# B&R Automation Studio project A2019059_Linka_Power_CP (part 58)

#### Main.st - Init, cyclic, exit code
```iecst
PROGRAM _INIT
	(* Insert code here *)

END_PROGRAM

PROGRAM _CYCLIC

	//Volanie funkcie SequenceControl//
	SequenceControl(SC:= SC_Devlink);

    //Mapovanie premenných//
    FTP_DMP_CAM17.STATUS.CisloPoruchy:= CisloAlarmu;
    FTP_DMP_CAM17.STATUS.AdresarPrazdny:= AdresarPrazdny;

    //Čísla alarmov//
    //1 - porucha otvorenia komunikacie z adresarom PLC
    //2 - porucha otvorenia komunikacie z adresarom Panasonic
    //3 - porucha načítania adresára kamery
    //4 - porucha zápisu najdených súborov
    //5 - porucha premenovania fotky
    //6 - porucha vytvorenia adresara na disku Panasonic
    //7 - porucha kopirovania fotky na server Panasonic
    //8 - porucha vymazania fotky v adresari kamery

    CASE SC_Devlink.Step OF

        0:
            SC_Devlink.StepName:= '0 - Nulovanie';
            FTP_DMP_CAM17.STATUS.KomunikaciaError:= FALSE;
            FTP_DMP_CAM17.STATUS.KomunikaciaUkoncena:= FALSE;
            PocetHladaniFotky:= 0;
            AdresarPrazdny:= FALSE;
            PocetNajdenychSuborov:= 0;
            PocetNajdenychAdresarov:= 0;
            PocetPremenovanychSuborov:= 1;
            PocetSkopirovanychSuborov:= 1;
            PocetVymazanychSuborov:= 1;
            i:= 0;
            SC_Devlink.Step:= 1;

        1:
            SC_Devlink.StepName:= '1 - Rozhodnutie o cinnosti';
            IF FTP_DMP_CAM17.CMD.OdosliFotku THEN
                CisloAlarmu:= 0;
                SC_Devlink.Step:= 10;
            ELSIF FTP_DMP_CAM17.CMD.VymazFotku THEN
                CisloAlarmu:= 0;
                SC_Devlink.Step:= 150;
            END_IF

        10:
            SC_Devlink.StepName:= '10 - Skopirovanie fotky do adresara DMP, otvorenie komunikacie z adresarom PLC';
            SC_Devlink.IdleTime.PT:= T#3s;
            SC_Devlink.AlarmTime.PT:= T#3s;

            DevLink_0.enable:= TRUE;
            DevLink_0.pDevice:= ADR('CAM17');
            DevLink_0.pParam:= ADR('/SIP=192.168.122.3 /PROTOCOL=ftp /USER=cam17 /PASSWORD=.cam17');
            DevLink_0();

            IF DevLink_0.enable THEN
                IF DevLink_0.status = 0 THEN
                    ID_Adresara1:= DevLink_0.handle;
                    SC_Devlink.ResetStep:= TRUE;
                    SC_Devlink.Step:= 15;//15
                ELSIF DevLink_0.status = 20730 THEN
                    ID_Adresara1:= DevLink_0.handle;
                    SC_Devlink.ResetStep:= TRUE;
                    SC_Devlink.Step:= 15;//15
                ELSIF DevLink_0.status = 65535 THEN
                    //BUSY//
                ELSE
                    CisloAlarmu:= 1;
                    FTP_DMP_CAM17.STATUS.KomunikaciaError:= TRUE;
                    SC_Devlink.ResetStep:= TRUE;
                    SC_Devlink.Step:= 13;
                END_IF
            END_IF

        13: SC_Devlink.StepName:= '13 - Skopirovanie fotky do adresara DMP, odpojenie od adresara PLC';
            SC_Devlink.IdleTime.PT:= T#3s;
            SC_Devlink.AlarmTime.PT:= T#3s;

            DevUnlink_0.enable:= TRUE;
            DevUnlink_0.handle:= ID_Adresara1;
            DevUnlink_0();

            IF DevUnlink_0.enable THEN
                IF DevUnlink_0.status = 0 THEN
                    SC_Devlink.ResetStep:= TRUE;
                    SC_Devlink.Step:= 100;
                ELSIF DevUnlink_0.status = 20731 THEN
                    SC_Devlink.ResetStep:= TRUE;
                    SC_Devlink.Step:= 100;
                ELSIF DevUnlink_0.status = 65535 THEN
                    //BUSY//
                ELSE
                    SC_Devlink.ResetStep:= TRUE;
                    SC_Devlink.Step:= 100;
                END_IF
            END_IF

        15:
            SC_Devlink.StepName:= '15 - Skopirovanie fotky do adresara DMP, otvorenie komunikacie z adresarom DMP';
            SC_Devlink.IdleTime.PT:= T#3s;
            SC_Devlink.AlarmTime.PT:= T#3s;

            DevLink_1.enable:= TRUE;
            DevLink_1.pDevice:= ADR('DMP_CAM17');
            DevLink_1.pParam:= ADR('/SIP=192.168.122.3 /PROTOCOL=ftp /USER=dmp_cam17 /PASSWORD=.dmp_cam17');
            DevLink_1();

            IF DevLink_1.enable THEN
                IF DevLink_1.status = 0 THEN
                    ID_Adresara2:= DevLink_0.handle;
                    SC_Devlink.ResetStep:= TRUE;
                    SC_Devlink.Step:= 20;
                ELSIF DevLink_1.status = 20730 THEN
                    ID_Adresara2:= DevLink_1.handle;
                    SC_Devlink.ResetStep:= TRUE;
                    SC_Devlink.Step:= 20;
                ELSIF DevLink_1.status = 65535 THEN
                    //BUSY//
                ELSE
                    CisloAlarmu:= 2;
                    FTP_DMP_CAM17.STATUS.KomunikaciaError:= TRUE;
                    SC_Devlink.ResetStep:= TRUE;
                    SC_Devlink.Step:= 18;
                END_IF
            END_IF

        18: SC_Devlink.StepName:= '18 - Skopirovanie fotky do adresara DMP, odpojenie od adresara DMP';
            SC_Devlink.IdleTime.PT:= T#3s;
            SC_Devlink.AlarmTime.PT:= T#3s;

            DevUnlink_1.enable:= TRUE;
            DevUnlink_1.handle:= ID_Adresara2;
            DevUnlink_1();

            IF DevUnlink_1.enable THEN
                IF DevUnlink_1.status = 0 THEN
                    SC_Devlink.ResetStep:= TRUE;
                    SC_Devlink.Step:= 100;
                ELSIF DevUnlink_1.status = 20731 THEN
                    SC_Devlink.ResetStep:= TRUE;
                    SC_Devlink.Step:= 100;
                ELSIF DevUnlink_1.status = 65535 THEN
                    //BUSY//
                ELSE
                    SC_Devlink.ResetStep:= TRUE;
                    SC_Devlink.Step:= 100;
                END_IF
            END_IF

        20:	SC_Devlink.StepName:= '20 - Skopirovanie fotky do adresara DMP, nacitanie adresara pred kopirovanim fotiek na server Panasonic';
            SC_Devlink.IdleTime.PT:= T#3s;
            SC_Devlink.AlarmTime.PT:= T#3s;

            DirInfo_0.enable:= TRUE;
            DirInfo_0.pDevice:= ADR('CAM17');
            DirInfo_0.pPath:= ADR('/');   //ak je nula tak číta všetky súbory a adresáre v koreni ak je "/Temp" tak číta všetky súbory a adresáre v adresári Temp//
            DirInfo_0();

            IF DirInfo_0.status = 0 THEN
                PocetNajdenychAdresarov:= DirInfo_0.dirnum;
                PocetNajdenychSuborov:= DirInfo_0.filenum;
                brsmemset(ADR(FileList[0]),0, SIZEOF(FileList));  //Vynulovanie pola stringov pre záznam adresárov a súborov
                SC_Devlink.ResetStep:= TRUE;
                SC_Devlink.Step:= 45;
            ELSIF DirInfo_0.status = 65535 THEN
                //BUSY//
            ELSIF DirInfo_0.status = 20723 THEN
                CisloAlarmu:= 3;
                FTP_DMP_CAM17.STATUS.KomunikaciaError:= TRUE;
                SC_Devlink.ResetStep:= TRUE;
                SC_Devlink.Step:= 100;
            ELSE
                CisloAlarmu:= 3;
                FTP_DMP_CAM17.STATUS.KomunikaciaError:= TRUE;
                SC_Devlink.ResetStep:= TRUE;
                SC_Devlink.Step:= 100;
            END_IF

        45: SC_Devlink.StepName:= '45 - Skopirovanie fotky do adresara DMP, zapis nazvou najdenych suborov do pola stringov';
            SC_Devlink.IdleTime.PT:= T#3s;
            SC_Devlink.AlarmTime.PT:= T#3s;

            DirRead_0.enable:= TRUE;
            DirRead_0.pDevice:= ADR('CAM17');
            DirRead_0.pPath:= ADR('/');   //ak je nula tak číta všetky súbory a adresáre v koreni ak je "/Temp" tak číta všetky súbory a adresáre v adresári Temp//
            DirRead_0.option:= fiFILE; //Zapíše súbory aj adresáre, ak je fiDIRECTORY zapíše len adresáre, ak je fiFILE tak zapíše len súbory//
            DirRead_0.entry:= i; //index zapisovania do pola//
            DirRead_0.pData:= ADR(ReadData);
            DirRead_0.data_len:= SIZEOF(ReadData);
            DirRead_0();

            IF DirRead_0.status = 0 THEN
                brsstrcpy(ADR(FileList[i]), ADR(ReadData.Filename[0])); //Uloženie názvou adresárov a súborov do pola stringov
                IF i< 100 THEN
                    i:= i + 1;
                END_IF
            ELSIF DirRead_0.status = 20702 THEN
                i:= 0;
                SC_Devlink.ResetStep:= TRUE;
                SC_Devlink.Step:= 48;
            ELSIF DirRead_0.status = 65535 THEN
                //BUSY//
            ELSE
                CisloAlarmu:= 4;
                FTP_DMP_CAM17.STATUS.KomunikaciaError:= TRUE;
                SC_Devlink.ResetStep:= TRUE;
                SC_Devlink.Step:= 100;
            END_IF

        48: SC_Devlink.StepName:= '48 - Skopirovanie fotky do adresara DMP, kopirovanie fotky do adresara DMP';
            SC_Devlink.IdleTime.PT:= T#3s;
            SC_Devlink.AlarmTime.PT:= T#3s;

            ZdrojKopirovaniaSuboru:= '';
            brsstrcat(ADR(ZdrojKopirovaniaSuboru),ADR('/'));
            brsstrcat(ADR(ZdrojKopirovaniaSuboru),ADR(FileList[i]));

            CielKopirovaniaSuboru:= '';
            brsstrcat(ADR(CielKopirovaniaSuboru),ADR('/'));
            brsstrcat(ADR(CielKopirovaniaSuboru),ADR(FileList[i]));

            FileCopy_0.enable:= TRUE;
            FileCopy_0.pSrcDev:= ADR('CAM17'); //Zdrojové zariadenie od kial sa kopíruje
            FileCopy_0.pSrc:= ADR(ZdrojKopirovaniaSuboru);
            FileCopy_0.pDestDev:= ADR('DMP_CAM17'); //Cielové zariadenie kam sa má súbor skopírovať
            FileCopy_0.pDest:= ADR(CielKopirovaniaSuboru);
            FileCopy_0();

            IF FileCopy_0.status = 0 THEN
                SC_Devlink.ResetStep:= TRUE;
                SC_Devlink.Step:= 50;
            ELSIF FileCopy_0.status = 65535 THEN
                //BUSY//
            ELSIF FileCopy_0.status = 20705 THEN
                SC_Devlink.ResetStep:= TRUE;
                SC_Devlink.Step:= 50;
            ELSIF FileCopy_0.status = 20708 THEN
                AdresarPrazdny:= TRUE;
                FTP_DMP_CAM17.STATUS.KomunikaciaUkoncena:= TRUE;
                SC_Devlink.ResetStep:= TRUE;
                SC_Devlink.Step:= 100;
            ELSE
                CisloAlarmu:= 7;
                FTP_DMP_CAM17.STATUS.KomunikaciaError:= TRUE;
                SC_Devlink.ResetStep:= TRUE;
                SC_Devlink.Step:= 100;
            END_IF

        50: SC_Devlink.StepName:= '50 - Skopirovanie fotky do adresara DMP, kontrola poctu skopirovanych suborov';
            SC_Devlink.IdleTime.PT:= T#3s;
            SC_Devlink.AlarmTime.PT:= T#3s;

            IF PocetSkopirovanychSuborov < PocetNajdenychSuborov THEN
                PocetSkopirovanychSuborov:= PocetSkopirovanychSuborov + 1;
                IF i< 100 THEN
                    i:= i + 1;
                END_IF
                SC_Devlink.ResetStep:= TRUE;
                SC_Devlink.Step:= 48;
            ELSE
                i:= 0;
                PocetNajdenychSuborov:= 0;
                PocetNajdenychAdresarov:= 0;
                FTP_DMP_CAM17.STATUS.KomunikaciaUkoncena:= TRUE;
                SC_Devlink.ResetStep:= TRUE;
                SC_Devlink.Step:= 100;
            END_IF

        100:
            SC_Devlink.StepName:= '100 - Skopirovanie fotky do adresara DMP, cakam na zrusenie prikazu odosli fotku';
            SC_Devlink.IdleTime.PT:= T#3s;
            SC_Devlink.AlarmTime.PT:= T#3s;

            IF NOT FTP_DMP_CAM17.CMD.OdosliFotku THEN
                SC_Devlink.ResetStep:= TRUE;
                SC_Devlink.Step:= 0;
            END_IF

            //**************************************Vymazanie fotky*************************************************//

        150:
            SC_Devlink.StepName:= '150 - Vymazanie fotky v adresari DMP, otvorenie komunikacie z adresarom DMP';
            SC_Devlink.IdleTime.PT:= T#3s;
            SC_Devlink.AlarmTime.PT:= T#3s;

            DevLink_0.enable:= TRUE;
            DevLink_0.pDevice:= ADR('DMP_CAM17');
            DevLink_0.pParam:= ADR('/SIP=192.168.122.3 /PROTOCOL=ftp /USER=dmp_cam17 /PASSWORD=.dmp_cam17');
            DevLink_0();

            IF DevLink_0.enable THEN
                IF DevLink_0.status = 0 THEN
                    ID_Adresara1:= DevLink_0.handle;
                    SC_Devlink.ResetStep:= TRUE;
                    SC_Devlink.Step:= 153;
                ELSIF DevLink_0.status = 20730 THEN
                    ID_Adresara1:= DevLink_0.handle;
                    SC_Devlink.ResetStep:= TRUE;
                    SC_Devlink.Step:= 153;
                ELSIF DevLink_0.status = 65535 THEN
                    //BUSY//
                ELSE
                    CisloAlarmu:= 1;
                    FTP_DMP_CAM17.STATUS.KomunikaciaError:= TRUE;
                    SC_Devlink.ResetStep:= TRUE;
                    SC_Devlink.Step:= 151;
                END_IF
            END_IF

        151: SC_Devlink.StepName:= '151 - Vymazanie fotky v adresari DMP, odpojenie od adresara DMP';
            SC_Devlink.IdleTime.PT:= T#3s;
            SC_Devlink.AlarmTime.PT:= T#3s;

            DevUnlink_0.enable:= TRUE;
            DevUnlink_0.handle:= ID_Adresara1;
            DevUnlink_0();

            IF DevUnlink_0.enable THEN
                IF DevUnlink_0.status = 0 THEN
                    SC_Devlink.ResetStep:= TRUE;
                    SC_Devlink.Step:= 200;
                ELSIF DevUnlink_0.status = 20731 THEN
                    SC_Devlink.ResetStep:= TRUE;
                    SC_Devlink.Step:= 200;
                ELSIF DevUnlink_0.status = 65535 THEN
                    //BUSY//
                ELSE
                    SC_Devlink.ResetStep:= TRUE;
                    SC_Devlink.Step:= 200;
                END_IF
            END_IF

        153:
            SC_Devlink.StepName:= '153 - Vymazanie fotky v adresari DMP, nacitanie adresara DMP pred vymazanim';
            SC_Devlink.IdleTime.PT:= T#3s;
            SC_Devlink.AlarmTime.PT:= T#3s;

            DirInfo_0.enable:= TRUE;
            DirInfo_0.pDevice:= ADR('DMP_CAM17');
            DirInfo_0.pPath:= ADR('/');   //ak je nula tak číta všetky súbory a adresáre v koreni ak je "/Temp" tak číta všetky súbory a adresáre v adresári Temp//
            DirInfo_0();

            IF DirInfo_0.status = 0 THEN
                PocetNajdenychAdresarov:= DirInfo_0.dirnum;
                PocetNajdenychSuborov:= DirInfo_0.filenum;
                brsmemset(ADR(FileList[0]),0, SIZEOF(FileList));  //Vynulovanie pola stringov pre záznam adresárov a súborov
                SC_Devlink.Step:= 155;
            ELSIF DirInfo_0.status = 65535 THEN
                //BUSY//
            ELSIF DirInfo_0.status = 20723 THEN
                CisloAlarmu:= 3;
                FTP_DMP_CAM17.STATUS.KomunikaciaError:= TRUE;
                SC_Devlink.ResetStep:= TRUE;
                SC_Devlink.Step:= 200;
            ELSE
                CisloAlarmu:= 3;
                FTP_DMP_CAM17.STATUS.KomunikaciaError:= TRUE;
                SC_Devlink.ResetStep:= TRUE;
                SC_Devlink.Step:= 200;
            END_IF

        155: SC_Devlink.StepName:= '155 - Vymazanie fotky v adresari DMP, zapis nazvou najdenych suborov do pola stringov';
            SC_Devlink.IdleTime.PT:= T#3s;
            SC_Devlink.AlarmTime.PT:= T#3s;

            DirRead_0.enable:= TRUE;
            DirRead_0.pDevice:= ADR('DMP_CAM17');
            DirRead_0.pPath:= ADR('/');   //ak je nula tak číta všetky súbory a adresáre v koreni ak je "/Temp" tak číta všetky súbory a adresáre v adresári Temp//
            DirRead_0.option:= fiFILE; //Zapíše súbory aj adresáre, ak je fiDIRECTORY zapíše len adresáre, ak je fiFILE tak zapíše len súbory//
            DirRead_0.entry:= i; //index zapisovania do pola//
            DirRead_0.pData:= ADR(ReadData);
            DirRead_0.data_len:= SIZEOF(ReadData);
            DirRead_0();

            IF DirRead_0.status = 0 THEN
                brsstrcpy(ADR(FileList[i]), ADR(ReadData.Filename[0])); //Uloženie názvou adresárov a súborov do pola stringov
				IF i< 100 THEN
					i:= i + 1;
				END_IF
            ELSIF DirRead_0.status = 20702 THEN
                i:= 0;
                SC_Devlink.ResetStep:= TRUE;
                SC_Devlink.Step:= 158;
            ELSIF DirRead_0.status = 65535 THEN
                //BUSY//
            ELSE
                CisloAlarmu:= 4;
                FTP_DMP_CAM17.STATUS.KomunikaciaError:= TRUE;
                SC_Devlink.ResetStep:= TRUE;
                SC_Devlink.Step:= 200;
            END_IF

        158: SC_Devlink.StepName:= '158 - Vymazanie fotky v adresari DMP, vymazanie suboru';
            SC_Devlink.IdleTime.PT:= T#3s;
            SC_Devlink.AlarmTime.PT:= T#3s;

            ZdrojKopirovaniaSuboru:= '';
            brsstrcat(ADR(ZdrojKopirovaniaSuboru),ADR('/'));
            brsstrcat(ADR(ZdrojKopirovaniaSuboru),ADR(FileList[i]));

            FileDelete_0.enable:= TRUE;
            FileDelete_0.pDevice:= ADR('DMP_CAM17');
            FileDelete_0.pName:= ADR(ZdrojKopirovaniaSuboru);
            FileDelete_0();

            IF FileDelete_0.status = 0 THEN
                SC_Devlink.ResetStep:= TRUE;
                SC_Devlink.Step:= 160;
            ELSIF FileDelete_0.status = 65535 THEN
                //BUSY//
            ELSIF FileDelete_0.status = 20708 THEN
                SC_Devlink.ResetStep:= TRUE;
                SC_Devlink.Step:= 160;
            ELSE
                CisloAlarmu:= 8;
                FTP_DMP_CAM17.STATUS.KomunikaciaError:= TRUE;
                SC_Devlink.ResetStep:= TRUE;
                SC_Devlink.Step:= 200;
            END_IF

        160:	SC_Devlink.StepName:= '160 - Vymazanie fotky v adresari DMP, kontrola poctu vymazanych suborov';
            SC_Devlink.IdleTime.PT:= T#3s;
            SC_Devlink.AlarmTime.PT:= T#3s;

            IF PocetVymazanychSuborov < PocetNajdenychSuborov THEN
                PocetVymazanychSuborov:= PocetVymazanychSuborov + 1;
                IF i< 100 THEN
                    i:= i + 1;
                END_IF
				SC_Devlink.ResetStep:= TRUE;
                SC_Devlink.Step:= 158;
            ELSE
                i:= 0;
                PocetNajdenychSuborov:= 0;
                PocetNajdenychAdresarov:= 0;
                FTP_DMP_CAM17.STATUS.KomunikaciaUkoncena:= TRUE;
                SC_Devlink.ResetStep:= TRUE;
                SC_Devlink.Step:= 200;
            END_IF

        200:
            SC_Devlink.StepName:= '200 - Vymazanie fotky v adresari DMP, cakam na zrusenie prikazu vymaz fotky';
            SC_Devlink.IdleTime.PT:= T#3s;
            SC_Devlink.AlarmTime.PT:= T#3s;

            IF NOT FTP_DMP_CAM17.CMD.VymazFotku THEN
                SC_Devlink.ResetStep:= TRUE;
                SC_Devlink.Step:= 0;
            END_IF

      END_CASE

END_PROGRAM

PROGRAM _EXIT
	(* Insert code here *)

END_PROGRAM
```

#### Variables.var - Local variables
```iecst
VAR
	SC_Devlink : SequenceControlTyp;
	DevLink_0 : DevLink;
	DevUnlink_0 : DevUnlink;
	DevLink_1 : DevLink;
	DevUnlink_1 : DevUnlink;
	DirInfo_0 : DirInfo;
	DirRead_0 : DirRead;
	FileRename_0 : FileRename;
	FileDelete_0 : FileDelete;
	FileCopy_0 : FileCopy;
	DirCreate_0 : DirCreate;
	i : UDINT;
	FileList : ARRAY[0..100] OF STRING[100];
	ReadData : fiDIR_READ_DATA; (*data-structure for command bDirRead*)
	ID_Adresara1 : UDINT;
	ID_Adresara2 : UDINT;
	PocetNajdenychAdresarov : UDINT;
	PocetNajdenychSuborov : UDINT;
	PocetPremenovanychSuborov : UDINT;
	PocetSkopirovanychSuborov : UDINT;
	PocetVymazanychSuborov : UDINT;
	StaryNazovSuboru : STRING[200];
	NovyNazovSuboru : STRING[200];
	ZdrojKopirovaniaSuboru : STRING[200];
	CielKopirovaniaSuboru : STRING[200];
	CisloAlarmu : USINT;
	AdresarPrazdny : BOOL;
	StruktNovehoNazvuSuboru : StrukturaNovehoNazvuSuboru_typ;
	StruktNovehoNazvuAdresara : StrukturaNovehoNazvuAdresara_typ;
	NazovAdresara_LINKA : STRING[50];
	NazovPodAdresara_PRACOVISKO : STRING[50];
	NazovPodAdresara_ROK : STRING[50];
	NazovPodAdresara_DATUM : STRING[50];
	PocetHladaniFotky : UDINT;
END_VAR
```

### Program Logical/MeranieTaktimePracovisk/TaktimeVytah_ST1 (IEC)

#### Main.st - Init, cyclic, exit code
```iecst
PROGRAM _INIT
	(* Insert code here *)

END_PROGRAM

PROGRAM _CYCLIC

    //Taktime pracoviska s presunom paletky//
    IF Taktime_Vytah_ST1.CMD.START_Merania_1 THEN

        Milisekundy_1:= Milisekundy_1 + 8;//Pretože je v taskovej triede 8ms tak prirátaváme + 8//

        IF Milisekundy_1 >= 1000 THEN
            Sekundy_1:= Sekundy_1 + 1;
            Milisekundy_1:= 0;
        END_IF

        IF Sekundy_1 >= 60 THEN
            Minuty_1:= Minuty_1 + 1;
            Sekundy_1:= 0;
        END_IF

        IF Minuty_1 >= 60 THEN
            Hodiny_1:= Hodiny_1 + 1;
            Minuty_1:= 0;
        END_IF

    END_IF

    IF NOT Taktime_Vytah_ST1.CMD.START_Merania_1 THEN
        Milisekundy_1:= 0;
        Sekundy_1:= 0;
        Minuty_1:= 0;
        Hodiny_1:= 0;
     END_IF

    IF Taktime_Vytah_ST1.CMD.ZAPIS_Hodnot_1 THEN
        Taktime_Vytah_ST1.OUTPUTS.NameraneHodiny_1:= Hodiny_1;
        Taktime_Vytah_ST1.OUTPUTS.NameraneMinuty_1:= Minuty_1;
        Taktime_Vytah_ST1.OUTPUTS.NameraneSekundy_1:= Sekundy_1;
        Milisekundy_1:= 0;
        Sekundy_1:= 0;
        Minuty_1:= 0;
        Hodiny_1:= 0;
        Taktime_Vytah_ST1.CMD.ZAPIS_Hodnot_1:= FALSE;
    END_IF

	IF Taktime_Vytah_ST1.CMD.STOP_Merania_1 THEN
		Taktime_Vytah_ST1.OUTPUTS.NameraneHodiny_1:= Hodiny_1;
		Taktime_Vytah_ST1.OUTPUTS.NameraneMinuty_1:= Minuty_1;
		Taktime_Vytah_ST1.OUTPUTS.NameraneSekundy_1:= Sekundy_1;
		Taktime_Vytah_ST1.CMD.START_Merania_1:= FALSE;
		Taktime_Vytah_ST1.CMD.STOP_Merania_1:= FALSE;
	END_IF

    //Taktime pracoviska bez presunu paletky//
    IF Taktime_Vytah_ST1.CMD.START_Merania_2 THEN

        Milisekundy_2:= Milisekundy_2 + 4;//Pretože je v taskovej triede 4ms tak prirátaváme + 4//

        IF Milisekundy_2 >= 1000 THEN
            Sekundy_2:= Sekundy_2 + 1;
            Milisekundy_2:= 0;
        END_IF

        IF Sekundy_2 >= 60 THEN
            Minuty_2:= Minuty_2 + 1;
            Sekundy_2:= 0;
        END_IF

        IF Minuty_2 >= 60 THEN
            Hodiny_2:= Hodiny_2 + 1;
            Minuty_2:= 0;
        END_IF

    END_IF

    IF NOT Taktime_Vytah_ST1.CMD.START_Merania_2 THEN
        Milisekundy_2:= 0;
        Sekundy_2:= 0;
        Minuty_2:= 0;
        Hodiny_2:= 0;
    END_IF

    IF Taktime_Vytah_ST1.CMD.ZAPIS_Hodnot_2 THEN
        Taktime_Vytah_ST1.OUTPUTS.NameraneHodiny_2:= Hodiny_2;
        Taktime_Vytah_ST1.OUTPUTS.NameraneMinuty_2:= Minuty_2;
        Taktime_Vytah_ST1.OUTPUTS.NameraneSekundy_2:= Sekundy_2;
        Milisekundy_2:= 0;
        Sekundy_2:= 0;
        Minuty_2:= 0;
        Hodiny_2:= 0;
        Taktime_Vytah_ST1.CMD.ZAPIS_Hodnot_2:= FALSE;
    END_IF

    IF Taktime_Vytah_ST1.CMD.STOP_Merania_2 THEN
		Taktime_Vytah_ST1.OUTPUTS.NameraneHodiny_2:= Hodiny_2;
		Taktime_Vytah_ST1.OUTPUTS.NameraneMinuty_2:= Minuty_2;
		Taktime_Vytah_ST1.OUTPUTS.NameraneSekundy_2:= Sekundy_2;
		Taktime_Vytah_ST1.CMD.START_Merania_2:= FALSE;
		Taktime_Vytah_ST1.CMD.STOP_Merania_2:= FALSE;
	END_IF

END_PROGRAM

PROGRAM _EXIT
	(* Insert code here *)

END_PROGRAM
```

#### Variables.var - Local variables
```iecst
VAR
	Milisekundy_1 : UINT;
	Sekundy_1 : UINT;
	Minuty_1 : UINT;
	Hodiny_1 : UINT;
	Milisekundy_2 : UINT;
	Sekundy_2 : UINT;
	Minuty_2 : UINT;
	Hodiny_2 : UINT;
END_VAR
```

### Program Logical/MeranieTaktimePracovisk/TaktimeSrobovanie_ST2 (IEC)

#### Main.st - Init, cyclic, exit code
```iecst
PROGRAM _INIT
	(* Insert code here *)

END_PROGRAM

PROGRAM _CYCLIC

    //Taktime pracoviska s presunom paletky//
    IF Taktime_Srobovanie_ST2.CMD.START_Merania_1 THEN

        Milisekundy_1:= Milisekundy_1 + 8;//Pretože je v taskovej triede 8ms tak prirátaváme + 8//

        IF Milisekundy_1 >= 1000 THEN
            Sekundy_1:= Sekundy_1 + 1;
            Milisekundy_1:= 0;
        END_IF

        IF Sekundy_1 >= 60 THEN
            Minuty_1:= Minuty_1 + 1;
            Sekundy_1:= 0;
        END_IF

        IF Minuty_1 >= 60 THEN
            Hodiny_1:= Hodiny_1 + 1;
            Minuty_1:= 0;
        END_IF

    END_IF

    IF NOT Taktime_Srobovanie_ST2.CMD.START_Merania_1 THEN
        Milisekundy_1:= 0;
        Sekundy_1:= 0;
        Minuty_1:= 0;
        Hodiny_1:= 0;
    END_IF

    IF Taktime_Srobovanie_ST2.CMD.ZAPIS_Hodnot_1 THEN
        Taktime_Srobovanie_ST2.OUTPUTS.NameraneHodiny_1:= Hodiny_1;
        Taktime_Srobovanie_ST2.OUTPUTS.NameraneMinuty_1:= Minuty_1;
        Taktime_Srobovanie_ST2.OUTPUTS.NameraneSekundy_1:= Sekundy_1;
        Taktime_Srobovanie_ST2.OUTPUTS.NameraneMilisekundy_1:= Milisekundy_1;
        Milisekundy_1:= 0;
        Sekundy_1:= 0;
        Minuty_1:= 0;
        Hodiny_1:= 0;
        Taktime_Srobovanie_ST2.CMD.ZAPIS_Hodnot_1:= FALSE;
    END_IF

	IF Taktime_Srobovanie_ST2.CMD.STOP_Merania_1 THEN
		Taktime_Srobovanie_ST2.OUTPUTS.NameraneHodiny_1:= Hodiny_1;
		Taktime_Srobovanie_ST2.OUTPUTS.NameraneMinuty_1:= Minuty_1;
		Taktime_Srobovanie_ST2.OUTPUTS.NameraneSekundy_1:= Sekundy_1;
		Taktime_Srobovanie_ST2.CMD.START_Merania_1:= FALSE;
		Taktime_Srobovanie_ST2.CMD.STOP_Merania_1:= FALSE;
	END_IF

    //Taktime pracoviska bez presunu paletky//
    IF Taktime_Srobovanie_ST2.CMD.START_Merania_2 THEN

        Milisekundy_2:= Milisekundy_2 + 4;//Pretože je v taskovej triede 4ms tak prirátaváme + 4//

        IF Milisekundy_2 >= 1000 THEN
            Sekundy_2:= Sekundy_2 + 1;
            Milisekundy_2:= 0;
        END_IF

        IF Sekundy_2 >= 60 THEN
            Minuty_2:= Minuty_2 + 1;
            Sekundy_2:= 0;
        END_IF

        IF Minuty_2 >= 60 THEN
            Hodiny_2:= Hodiny_2 + 1;
            Minuty_2:= 0;
        END_IF

    END_IF

    IF NOT Taktime_Srobovanie_ST2.CMD.START_Merania_2 THEN
        Milisekundy_2:= 0;
        Sekundy_2:= 0;
        Minuty_2:= 0;
        Hodiny_2:= 0;
    END_IF

    IF Taktime_Srobovanie_ST2.CMD.ZAPIS_Hodnot_2 THEN
        Taktime_Srobovanie_ST2.OUTPUTS.NameraneHodiny_2:= Hodiny_2;
        Taktime_Srobovanie_ST2.OUTPUTS.NameraneMinuty_2:= Minuty_2;
        Taktime_Srobovanie_ST2.OUTPUTS.NameraneSekundy_2:= Sekundy_2;
        Taktime_Srobovanie_ST2.OUTPUTS.NameraneMilisekundy_2:= Milisekundy_2;
        Milisekundy_2:= 0;
        Sekundy_2:= 0;
        Minuty_2:= 0;
        Hodiny_2:= 0;
        Taktime_Srobovanie_ST2.CMD.ZAPIS_Hodnot_2:= FALSE;
    END_IF

	IF Taktime_Srobovanie_ST2.CMD.STOP_Merania_2 THEN
		Taktime_Srobovanie_ST2.OUTPUTS.NameraneHodiny_2:= Hodiny_2;
		Taktime_Srobovanie_ST2.OUTPUTS.NameraneMinuty_2:= Minuty_2;
		Taktime_Srobovanie_ST2.OUTPUTS.NameraneSekundy_2:= Sekundy_2;
		Taktime_Srobovanie_ST2.CMD.START_Merania_2:= FALSE;
		Taktime_Srobovanie_ST2.CMD.STOP_Merania_2:= FALSE;
	END_IF

END_PROGRAM

PROGRAM _EXIT
	(* Insert code here *)

END_PROGRAM
```

#### Variables.var - Local variables
```iecst
VAR
	Milisekundy_1 : UINT;
	Sekundy_1 : UINT;
	Minuty_1 : UINT;
	Hodiny_1 : UINT;
	Milisekundy_2 : UINT;
	Sekundy_2 : UINT;
	Minuty_2 : UINT;
	Hodiny_2 : UINT;
END_VAR
```

### Program Logical/MeranieTaktimePracovisk/TaktimeZaklTesnenia_ST3 (IEC)

#### Main.st - Init, cyclic, exit code
```iecst
PROGRAM _INIT
	(* Insert code here *)

END_PROGRAM

PROGRAM _CYCLIC

    //Taktime pracoviska s presunom paletky//
    IF Taktime_ZakladacTesnenia_ST3.CMD.START_Merania_1 THEN

        Milisekundy_1:= Milisekundy_1 + 8;//Pretože je v taskovej triede 8ms tak prirátaváme + 8//

        IF Milisekundy_1 >= 1000 THEN
            Sekundy_1:= Sekundy_1 + 1;
            Milisekundy_1:= 0;
        END_IF

        IF Sekundy_1 >= 60 THEN
            Minuty_1:= Minuty_1 + 1;
            Sekundy_1:= 0;
        END_IF

        IF Minuty_1 >= 60 THEN
            Hodiny_1:= Hodiny_1 + 1;
            Minuty_1:= 0;
        END_IF

    END_IF

    IF NOT Taktime_ZakladacTesnenia_ST3.CMD.START_Merania_1 THEN
        Milisekundy_1:= 0;
        Sekundy_1:= 0;
        Minuty_1:= 0;
        Hodiny_1:= 0;
    END_IF

    IF Taktime_ZakladacTesnenia_ST3.CMD.ZAPIS_Hodnot_1 THEN
        Taktime_ZakladacTesnenia_ST3.OUTPUTS.NameraneHodiny_1:= Hodiny_1;
        Taktime_ZakladacTesnenia_ST3.OUTPUTS.NameraneMinuty_1:= Minuty_1;
        Taktime_ZakladacTesnenia_ST3.OUTPUTS.NameraneSekundy_1:= Sekundy_1;
        Milisekundy_1:= 0;
        Sekundy_1:= 0;
        Minuty_1:= 0;
        Hodiny_1:= 0;
        Taktime_ZakladacTesnenia_ST3.CMD.ZAPIS_Hodnot_1:= FALSE;
    END_IF

	IF Taktime_ZakladacTesnenia_ST3.CMD.STOP_Merania_1 THEN
		Taktime_ZakladacTesnenia_ST3.OUTPUTS.NameraneHodiny_1:= Hodiny_1;
		Taktime_ZakladacTesnenia_ST3.OUTPUTS.NameraneMinuty_1:= Minuty_1;
		Taktime_ZakladacTesnenia_ST3.OUTPUTS.NameraneSekundy_1:= Sekundy_1;
		Taktime_ZakladacTesnenia_ST3.CMD.START_Merania_1:= FALSE;
		Taktime_ZakladacTesnenia_ST3.CMD.STOP_Merania_1:= FALSE;
	END_IF

    //Taktime pracoviska bez presunu paletky//
    IF Taktime_ZakladacTesnenia_ST3.CMD.START_Merania_2 THEN

        Milisekundy_2:= Milisekundy_2 + 4;//Pretože je v taskovej triede 4ms tak prirátaváme + 4//

        IF Milisekundy_2 >= 1000 THEN
            Sekundy_2:= Sekundy_2 + 1;
            Milisekundy_2:= 0;
        END_IF

        IF Sekundy_2 >= 60 THEN
            Minuty_2:= Minuty_2 + 1;
            Sekundy_2:= 0;
        END_IF

        IF Minuty_2 >= 60 THEN
            Hodiny_2:= Hodiny_2 + 1;
            Minuty_2:= 0;
        END_IF

    END_IF

    IF NOT Taktime_ZakladacTesnenia_ST3.CMD.START_Merania_2 THEN
        Milisekundy_2:= 0;
        Sekundy_2:= 0;
        Minuty_2:= 0;
        Hodiny_2:= 0;
    END_IF

    IF Taktime_ZakladacTesnenia_ST3.CMD.ZAPIS_Hodnot_2 THEN
        Taktime_ZakladacTesnenia_ST3.OUTPUTS.NameraneHodiny_2:= Hodiny_2;
        Taktime_ZakladacTesnenia_ST3.OUTPUTS.NameraneMinuty_2:= Minuty_2;
        Taktime_ZakladacTesnenia_ST3.OUTPUTS.NameraneSekundy_2:= Sekundy_2;
        Milisekundy_2:= 0;
        Sekundy_2:= 0;
        Minuty_2:= 0;
        Hodiny_2:= 0;
        Taktime_ZakladacTesnenia_ST3.CMD.ZAPIS_Hodnot_2:= FALSE;
    END_IF

	IF Taktime_ZakladacTesnenia_ST3.CMD.STOP_Merania_2 THEN
		Taktime_ZakladacTesnenia_ST3.OUTPUTS.NameraneHodiny_2:= Hodiny_2;
		Taktime_ZakladacTesnenia_ST3.OUTPUTS.NameraneMinuty_2:= Minuty_2;
		Taktime_ZakladacTesnenia_ST3.OUTPUTS.NameraneSekundy_2:= Sekundy_2;
		Taktime_ZakladacTesnenia_ST3.CMD.START_Merania_2:= FALSE;
		Taktime_ZakladacTesnenia_ST3.CMD.STOP_Merania_2:= FALSE;
	END_IF

END_PROGRAM

PROGRAM _EXIT
	(* Insert code here *)

END_PROGRAM
```

#### Variables.var - Local variables
```iecst
VAR
	Milisekundy_1 : UINT;
	Sekundy_1 : UINT;
	Minuty_1 : UINT;
	Hodiny_1 : UINT;
	Milisekundy_2 : UINT;
	Sekundy_2 : UINT;
	Minuty_2 : UINT;
	Hodiny_2 : UINT;
END_VAR
```

### Program Logical/MeranieTaktimePracovisk/TaktimeMaticovacka_ST4 (IEC)

#### Main.st - Init, cyclic, exit code
```iecst
PROGRAM _INIT
	(* Insert code here *)

END_PROGRAM

PROGRAM _CYCLIC

     //Taktime pracoviska s presunom paletky//
    IF Taktime_Maticovacka_ST4.CMD.START_Merania_1 THEN

        Milisekundy_1:= Milisekundy_1 + 8;//Pretože je v taskovej triede 8ms tak prirátaváme + 8//

        IF Milisekundy_1 >= 1000 THEN
            Sekundy_1:= Sekundy_1 + 1;
            Milisekundy_1:= 0;
        END_IF

        IF Sekundy_1 >= 60 THEN
            Minuty_1:= Minuty_1 + 1;
            Sekundy_1:= 0;
        END_IF

        IF Minuty_1 >= 60 THEN
            Hodiny_1:= Hodiny_1 + 1;
            Minuty_1:= 0;
        END_IF

    END_IF

    IF NOT Taktime_Maticovacka_ST4.CMD.START_Merania_1 THEN
        Milisekundy_1:= 0;
        Sekundy_1:= 0;
        Minuty_1:= 0;
        Hodiny_1:= 0;
    END_IF

    IF Taktime_Maticovacka_ST4.CMD.ZAPIS_Hodnot_1 THEN
        Taktime_Maticovacka_ST4.OUTPUTS.NameraneHodiny_1:= Hodiny_1;
        Taktime_Maticovacka_ST4.OUTPUTS.NameraneMinuty_1:= Minuty_1;
        Taktime_Maticovacka_ST4.OUTPUTS.NameraneSekundy_1:= Sekundy_1;
        Milisekundy_1:= 0;
        Sekundy_1:= 0;
        Minuty_1:= 0;
        Hodiny_1:= 0;
        Taktime_Maticovacka_ST4.CMD.ZAPIS_Hodnot_1:= FALSE;
    END_IF

	IF Taktime_Maticovacka_ST4.CMD.STOP_Merania_1 THEN
		Taktime_Maticovacka_ST4.OUTPUTS.NameraneHodiny_1:= Hodiny_1;
		Taktime_Maticovacka_ST4.OUTPUTS.NameraneMinuty_1:= Minuty_1;
		Taktime_Maticovacka_ST4.OUTPUTS.NameraneSekundy_1:= Sekundy_1;
		Taktime_Maticovacka_ST4.CMD.START_Merania_1:= FALSE;
		Taktime_Maticovacka_ST4.CMD.STOP_Merania_1:= FALSE;
	END_IF

    //Taktime pracoviska bez presunu paletky//
    IF Taktime_Maticovacka_ST4.CMD.START_Merania_2 THEN

        Milisekundy_2:= Milisekundy_2 + 4;//Pretože je v taskovej triede 4ms tak prirátaváme + 4//

        IF Milisekundy_2 >= 1000 THEN
            Sekundy_2:= Sekundy_2 + 1;
            Milisekundy_2:= 0;
        END_IF

        IF Sekundy_2 >= 60 THEN
            Minuty_2:= Minuty_2 + 1;
            Sekundy_2:= 0;
        END_IF

        IF Minuty_2 >= 60 THEN
            Hodiny_2:= Hodiny_2 + 1;
            Minuty_2:= 0;
        END_IF

    END_IF

    IF NOT Taktime_Maticovacka_ST4.CMD.START_Merania_2 THEN
        Milisekundy_2:= 0;
        Sekundy_2:= 0;
        Minuty_2:= 0;
        Hodiny_2:= 0;
    END_IF

    IF Taktime_Maticovacka_ST4.CMD.ZAPIS_Hodnot_2 THEN
        Taktime_Maticovacka_ST4.OUTPUTS.NameraneHodiny_2:= Hodiny_2;
        Taktime_Maticovacka_ST4.OUTPUTS.NameraneMinuty_2:= Minuty_2;
        Taktime_Maticovacka_ST4.OUTPUTS.NameraneSekundy_2:= Sekundy_2;
        Milisekundy_2:= 0;
        Sekundy_2:= 0;
        Minuty_2:= 0;
        Hodiny_2:= 0;
        Taktime_Maticovacka_ST4.CMD.ZAPIS_Hodnot_2:= FALSE;
    END_IF

	IF Taktime_Maticovacka_ST4.CMD.STOP_Merania_2 THEN
		Taktime_Maticovacka_ST4.OUTPUTS.NameraneHodiny_2:= Hodiny_2;
		Taktime_Maticovacka_ST4.OUTPUTS.NameraneMinuty_2:= Minuty_2;
		Taktime_Maticovacka_ST4.OUTPUTS.NameraneSekundy_2:= Sekundy_2;
		Taktime_Maticovacka_ST4.CMD.START_Merania_2:= FALSE;
		Taktime_Maticovacka_ST4.CMD.STOP_Merania_2:= FALSE;
	END_IF

END_PROGRAM

PROGRAM _EXIT
	(* Insert code here *)

END_PROGRAM
```

#### Variables.var - Local variables
```iecst
VAR
	Milisekundy_1 : UINT;
	Sekundy_1 : UINT;
	Minuty_1 : UINT;
	Hodiny_1 : UINT;
	Milisekundy_2 : UINT;
	Sekundy_2 : UINT;
	Minuty_2 : UINT;
	Hodiny_2 : UINT;
END_VAR
```

### Program Logical/MeranieTaktimePracovisk/TaktimeSrobovanie_ST5 (IEC)

#### Main.st - Init, cyclic, exit code
```iecst
PROGRAM _INIT
	(* Insert code here *)

END_PROGRAM

PROGRAM _CYCLIC

    //Taktime pracoviska s presunom paletky//
    IF Taktime_Srobovanie_ST5.CMD.START_Merania_1 THEN

        Milisekundy_1:= Milisekundy_1 + 8;//Pretože je v taskovej triede 8ms tak prirátaváme + 8//

        IF Milisekundy_1 >= 1000 THEN
            Sekundy_1:= Sekundy_1 + 1;
            Milisekundy_1:= 0;
        END_IF

        IF Sekundy_1 >= 60 THEN
            Minuty_1:= Minuty_1 + 1;
            Sekundy_1:= 0;
        END_IF

        IF Minuty_1 >= 60 THEN
            Hodiny_1:= Hodiny_1 + 1;
            Minuty_1:= 0;
        END_IF

    END_IF

    IF NOT Taktime_Srobovanie_ST5.CMD.START_Merania_1 THEN
        Milisekundy_1:= 0;
        Sekundy_1:= 0;
        Minuty_1:= 0;
        Hodiny_1:= 0;
    END_IF

    IF Taktime_Srobovanie_ST5.CMD.ZAPIS_Hodnot_1 THEN
        Taktime_Srobovanie_ST5.OUTPUTS.NameraneHodiny_1:= Hodiny_1;
        Taktime_Srobovanie_ST5.OUTPUTS.NameraneMinuty_1:= Minuty_1;
        Taktime_Srobovanie_ST5.OUTPUTS.NameraneSekundy_1:= Sekundy_1;
        Milisekundy_1:= 0;
        Sekundy_1:= 0;
        Minuty_1:= 0;
        Hodiny_1:= 0;
        Taktime_Srobovanie_ST5.CMD.ZAPIS_Hodnot_1:= FALSE;
    END_IF

	IF Taktime_Srobovanie_ST5.CMD.STOP_Merania_1 THEN
		Taktime_Srobovanie_ST5.OUTPUTS.NameraneHodiny_1:= Hodiny_1;
		Taktime_Srobovanie_ST5.OUTPUTS.NameraneMinuty_1:= Minuty_1;
		Taktime_Srobovanie_ST5.OUTPUTS.NameraneSekundy_1:= Sekundy_1;
		Taktime_Srobovanie_ST5.CMD.START_Merania_1:= FALSE;
		Taktime_Srobovanie_ST5.CMD.STOP_Merania_1:= FALSE;
	END_IF

    //Taktime pracoviska bez presunu paletky//
    IF Taktime_Srobovanie_ST5.CMD.START_Merania_2 THEN

        Milisekundy_2:= Milisekundy_2 + 4;//Pretože je v taskovej triede 4ms tak prirátaváme + 4//

        IF Milisekundy_2 >= 1000 THEN
            Sekundy_2:= Sekundy_2 + 1;
            Milisekundy_2:= 0;
        END_IF

        IF Sekundy_2 >= 60 THEN
            Minuty_2:= Minuty_2 + 1;
            Sekundy_2:= 0;
        END_IF

        IF Minuty_2 >= 60 THEN
            Hodiny_2:= Hodiny_2 + 1;
            Minuty_2:= 0;
        END_IF

    END_IF

    IF NOT Taktime_Srobovanie_ST5.CMD.START_Merania_2 THEN
        Milisekundy_2:= 0;
        Sekundy_2:= 0;
        Minuty_2:= 0;
        Hodiny_2:= 0;
    END_IF

    IF Taktime_Srobovanie_ST5.CMD.ZAPIS_Hodnot_2 THEN
        Taktime_Srobovanie_ST5.OUTPUTS.NameraneHodiny_2:= Hodiny_2;
        Taktime_Srobovanie_ST5.OUTPUTS.NameraneMinuty_2:= Minuty_2;
        Taktime_Srobovanie_ST5.OUTPUTS.NameraneSekundy_2:= Sekundy_2;
        Milisekundy_2:= 0;
        Sekundy_2:= 0;
        Minuty_2:= 0;
        Hodiny_2:= 0;
        Taktime_Srobovanie_ST5.CMD.ZAPIS_Hodnot_2:= FALSE;
    END_IF

	IF Taktime_Srobovanie_ST5.CMD.STOP_Merania_2 THEN
		Taktime_Srobovanie_ST5.OUTPUTS.NameraneHodiny_2:= Hodiny_2;
		Taktime_Srobovanie_ST5.OUTPUTS.NameraneMinuty_2:= Minuty_2;
		Taktime_Srobovanie_ST5.OUTPUTS.NameraneSekundy_2:= Sekundy_2;
		Taktime_Srobovanie_ST5.CMD.START_Merania_2:= FALSE;
		Taktime_Srobovanie_ST5.CMD.STOP_Merania_2:= FALSE;
	END_IF

END_PROGRAM

PROGRAM _EXIT
	(* Insert code here *)

END_PROGRAM
```

#### Variables.var - Local variables
```iecst
VAR
	Milisekundy_1 : UINT;
	Sekundy_1 : UINT;
	Minuty_1 : UINT;
	Hodiny_1 : UINT;
	Milisekundy_2 : UINT;
	Sekundy_2 : UINT;
	Minuty_2 : UINT;
	Hodiny_2 : UINT;
END_VAR
```

### Program Logical/MeranieTaktimePracovisk/TaktimeZvaranie_ST6 (IEC)

#### Main.st - Init, cyclic, exit code
```iecst
PROGRAM _INIT
	(* Insert code here *)

END_PROGRAM

PROGRAM _CYCLIC

    //Taktime pracoviska s presunom paletky//
    IF Taktime_Zvaranie_ST6.CMD.START_Merania_1 THEN

        Milisekundy_1:= Milisekundy_1 + 8;//Pretože je v taskovej triede 8ms tak prirátaváme + 8//

        IF Milisekundy_1 >= 1000 THEN
            Sekundy_1:= Sekundy_1 + 1;
            Milisekundy_1:= 0;
        END_IF

        IF Sekundy_1 >= 60 THEN
            Minuty_1:= Minuty_1 + 1;
            Sekundy_1:= 0;
        END_IF

        IF Minuty_1 >= 60 THEN
            Hodiny_1:= Hodiny_1 + 1;
            Minuty_1:= 0;
        END_IF

    END_IF

    IF NOT Taktime_Zvaranie_ST6.CMD.START_Merania_1 THEN
        Milisekundy_1:= 0;
        Sekundy_1:= 0;
        Minuty_1:= 0;
        Hodiny_1:= 0;
    END_IF

    IF Taktime_Zvaranie_ST6.CMD.ZAPIS_Hodnot_1 THEN
        Taktime_Zvaranie_ST6.OUTPUTS.NameraneHodiny_1:= Hodiny_1;
        Taktime_Zvaranie_ST6.OUTPUTS.NameraneMinuty_1:= Minuty_1;
        Taktime_Zvaranie_ST6.OUTPUTS.NameraneSekundy_1:= Sekundy_1;
        Milisekundy_1:= 0;
        Sekundy_1:= 0;
        Minuty_1:= 0;
        Hodiny_1:= 0;
        Taktime_Zvaranie_ST6.CMD.ZAPIS_Hodnot_1:= FALSE;
    END_IF

	IF Taktime_Zvaranie_ST6.CMD.STOP_Merania_1 THEN
		Taktime_Zvaranie_ST6.OUTPUTS.NameraneHodiny_1:= Hodiny_1;
		Taktime_Zvaranie_ST6.OUTPUTS.NameraneMinuty_1:= Minuty_1;
		Taktime_Zvaranie_ST6.OUTPUTS.NameraneSekundy_1:= Sekundy_1;
		Taktime_Zvaranie_ST6.CMD.START_Merania_1:= FALSE;
		Taktime_Zvaranie_ST6.CMD.STOP_Merania_1:= FALSE;
	END_IF

    //Taktime pracoviska bez presunu paletky//
    IF Taktime_Zvaranie_ST6.CMD.START_Merania_2 THEN

        Milisekundy_2:= Milisekundy_2 + 4;//Pretože je v taskovej triede 4ms tak prirátaváme + 4//

        IF Milisekundy_2 >= 1000 THEN
            Sekundy_2:= Sekundy_2 + 1;
            Milisekundy_2:= 0;
        END_IF

        IF Sekundy_2 >= 60 THEN
            Minuty_2:= Minuty_2 + 1;
            Sekundy_2:= 0;
        END_IF

        IF Minuty_2 >= 60 THEN
            Hodiny_2:= Hodiny_2 + 1;
            Minuty_2:= 0;
        END_IF

    END_IF

    IF NOT Taktime_Zvaranie_ST6.CMD.START_Merania_2 THEN
        Milisekundy_2:= 0;
        Sekundy_2:= 0;
        Minuty_2:= 0;
        Hodiny_2:= 0;
    END_IF

    IF Taktime_Zvaranie_ST6.CMD.ZAPIS_Hodnot_2 THEN
        Taktime_Zvaranie_ST6.OUTPUTS.NameraneHodiny_2:= Hodiny_2;
        Taktime_Zvaranie_ST6.OUTPUTS.NameraneMinuty_2:= Minuty_2;
        Taktime_Zvaranie_ST6.OUTPUTS.NameraneSekundy_2:= Sekundy_2;
        Milisekundy_2:= 0;
        Sekundy_2:= 0;
        Minuty_2:= 0;
        Hodiny_2:= 0;
        Taktime_Zvaranie_ST6.CMD.ZAPIS_Hodnot_2:= FALSE;
    END_IF

	IF Taktime_Zvaranie_ST6.CMD.STOP_Merania_2 THEN
		Taktime_Zvaranie_ST6.OUTPUTS.NameraneHodiny_2:= Hodiny_2;
		Taktime_Zvaranie_ST6.OUTPUTS.NameraneMinuty_2:= Minuty_2;
		Taktime_Zvaranie_ST6.OUTPUTS.NameraneSekundy_2:= Sekundy_2;
		Taktime_Zvaranie_ST6.CMD.START_Merania_2:= FALSE;
		Taktime_Zvaranie_ST6.CMD.STOP_Merania_2:= FALSE;
	END_IF

END_PROGRAM

PROGRAM _EXIT
	(* Insert code here *)

END_PROGRAM
```

#### Variables.var - Local variables
```iecst
VAR
	Milisekundy_1 : UINT;
	Sekundy_1 : UINT;
	Minuty_1 : UINT;
	Hodiny_1 : UINT;
	Milisekundy_2 : UINT;
	Sekundy_2 : UINT;
	Minuty_2 : UINT;
	Hodiny_2 : UINT;
END_VAR
```

### Program Logical/MeranieTaktimePracovisk/Taktime_Srobovanie_ST7 (IEC)

#### Main.st - Init, cyclic, exit code
```iecst
PROGRAM _INIT
	(* Insert code here *)

END_PROGRAM

PROGRAM _CYCLIC

    //Taktime pracoviska s presunom paletky//
    IF Taktime_Srobovanie_ST7.CMD.START_Merania_1 THEN

        Milisekundy_1:= Milisekundy_1 + 8;//Pretože je v taskovej triede 8ms tak prirátaváme + 8//

        IF Milisekundy_1 >= 1000 THEN
            Sekundy_1:= Sekundy_1 + 1;
            Milisekundy_1:= 0;
        END_IF

        IF Sekundy_1 >= 60 THEN
            Minuty_1:= Minuty_1 + 1;
            Sekundy_1:= 0;
        END_IF

        IF Minuty_1 >= 60 THEN
            Hodiny_1:= Hodiny_1 + 1;
            Minuty_1:= 0;
        END_IF

    END_IF

    IF NOT Taktime_Srobovanie_ST7.CMD.START_Merania_1 THEN
        Milisekundy_1:= 0;
        Sekundy_1:= 0;
        Minuty_1:= 0;
        Hodiny_1:= 0;
    END_IF

    IF Taktime_Srobovanie_ST7.CMD.ZAPIS_Hodnot_1 THEN
        Taktime_Srobovanie_ST7.OUTPUTS.NameraneHodiny_1:= Hodiny_1;
        Taktime_Srobovanie_ST7.OUTPUTS.NameraneMinuty_1:= Minuty_1;
        Taktime_Srobovanie_ST7.OUTPUTS.NameraneSekundy_1:= Sekundy_1;
        Milisekundy_1:= 0;
        Sekundy_1:= 0;
        Minuty_1:= 0;
        Hodiny_1:= 0;
        Taktime_Srobovanie_ST7.CMD.ZAPIS_Hodnot_1:= FALSE;
    END_IF

	IF Taktime_Srobovanie_ST7.CMD.STOP_Merania_1 THEN
		Taktime_Srobovanie_ST7.OUTPUTS.NameraneHodiny_1:= Hodiny_1;
		Taktime_Srobovanie_ST7.OUTPUTS.NameraneMinuty_1:= Minuty_1;
		Taktime_Srobovanie_ST7.OUTPUTS.NameraneSekundy_1:= Sekundy_1;
		Taktime_Srobovanie_ST7.CMD.START_Merania_1:= FALSE;
		Taktime_Srobovanie_ST7.CMD.STOP_Merania_1:= FALSE;
	END_IF

    //Taktime pracoviska bez presunu paletky//
    IF Taktime_Srobovanie_ST7.CMD.START_Merania_2 THEN

        Milisekundy_2:= Milisekundy_2 + 4;//Pretože je v taskovej triede 4ms tak prirátaváme + 4//

        IF Milisekundy_2 >= 1000 THEN
            Sekundy_2:= Sekundy_2 + 1;
            Milisekundy_2:= 0;
        END_IF

        IF Sekundy_2 >= 60 THEN
            Minuty_2:= Minuty_2 + 1;
            Sekundy_2:= 0;
        END_IF

        IF Minuty_2 >= 60 THEN
            Hodiny_2:= Hodiny_2 + 1;
            Minuty_2:= 0;
        END_IF

    END_IF

    IF NOT Taktime_Srobovanie_ST7.CMD.START_Merania_2 THEN
        Milisekundy_2:= 0;
        Sekundy_2:= 0;
        Minuty_2:= 0;
        Hodiny_2:= 0;
    END_IF

    IF Taktime_Srobovanie_ST7.CMD.ZAPIS_Hodnot_2 THEN
        Taktime_Srobovanie_ST7.OUTPUTS.NameraneHodiny_2:= Hodiny_2;
        Taktime_Srobovanie_ST7.OUTPUTS.NameraneMinuty_2:= Minuty_2;
        Taktime_Srobovanie_ST7.OUTPUTS.NameraneSekundy_2:= Sekundy_2;
        Milisekundy_2:= 0;
        Sekundy_2:= 0;
        Minuty_2:= 0;
        Hodiny_2:= 0;
        Taktime_Srobovanie_ST7.CMD.ZAPIS_Hodnot_2:= FALSE;
    END_IF

	IF Taktime_Srobovanie_ST7.CMD.STOP_Merania_2 THEN
		Taktime_Srobovanie_ST7.OUTPUTS.NameraneHodiny_2:= Hodiny_2;
		Taktime_Srobovanie_ST7.OUTPUTS.NameraneMinuty_2:= Minuty_2;
		Taktime_Srobovanie_ST7.OUTPUTS.NameraneSekundy_2:= Sekundy_2;
		Taktime_Srobovanie_ST7.CMD.START_Merania_2:= FALSE;
		Taktime_Srobovanie_ST7.CMD.STOP_Merania_2:= FALSE;
	END_IF

END_PROGRAM

PROGRAM _EXIT
	(* Insert code here *)

END_PROGRAM
```

#### Variables.var - Local variables
```iecst
VAR
	Milisekundy_1 : UINT;
	Sekundy_1 : UINT;
	Minuty_1 : UINT;
	Hodiny_1 : UINT;
	Milisekundy_2 : UINT;
	Sekundy_2 : UINT;
	Minuty_2 : UINT;
	Hodiny_2 : UINT;
END_VAR
```

### Program Logical/MeranieTaktimePracovisk/Taktime_LeakageTestA_ST8A (IEC)

#### Main.st - Init, cyclic, exit code
```iecst
PROGRAM _INIT
	(* Insert code here *)

END_PROGRAM

PROGRAM _CYCLIC

        //Taktime pracoviska s presunom paletky//
	IF Taktime_LeakageTestA_ST8A.CMD.START_Merania_1 THEN

		Milisekundy_1:= Milisekundy_1 + 8;//Pretože je v taskovej triede 8ms tak prirátaváme + 8//

		IF Milisekundy_1 >= 1000 THEN
			Sekundy_1:= Sekundy_1 + 1;
			Milisekundy_1:= 0;
		END_IF

		IF Sekundy_1 >= 60 THEN
			Minuty_1:= Minuty_1 + 1;
			Sekundy_1:= 0;
		END_IF

		IF Minuty_1 >= 60 THEN
			Hodiny_1:= Hodiny_1 + 1;
			Minuty_1:= 0;
		END_IF

	END_IF

	IF NOT Taktime_LeakageTestA_ST8A.CMD.START_Merania_1 THEN
		Milisekundy_1:= 0;
		Sekundy_1:= 0;
		Minuty_1:= 0;
		Hodiny_1:= 0;
	END_IF

	IF Taktime_LeakageTestA_ST8A.CMD.ZAPIS_Hodnot_1 THEN
		Taktime_LeakageTestA_ST8A.OUTPUTS.NameraneHodiny_1:= Hodiny_1;
		Taktime_LeakageTestA_ST8A.OUTPUTS.NameraneMinuty_1:= Minuty_1;
		Taktime_LeakageTestA_ST8A.OUTPUTS.NameraneSekundy_1:= Sekundy_1;
		Milisekundy_1:= 0;
		Sekundy_1:= 0;
		Minuty_1:= 0;
		Hodiny_1:= 0;
		Taktime_LeakageTestA_ST8A.CMD.ZAPIS_Hodnot_1:= FALSE;
	END_IF

	IF Taktime_LeakageTestA_ST8A.CMD.STOP_Merania_1 THEN
		Taktime_LeakageTestA_ST8A.OUTPUTS.NameraneHodiny_1:= Hodiny_1;
		Taktime_LeakageTestA_ST8A.OUTPUTS.NameraneMinuty_1:= Minuty_1;
		Taktime_LeakageTestA_ST8A.OUTPUTS.NameraneSekundy_1:= Sekundy_1;
		Taktime_LeakageTestA_ST8A.CMD.START_Merania_1:= FALSE;
		Taktime_LeakageTestA_ST8A.CMD.STOP_Merania_1:= FALSE;
	END_IF

	//Taktime pracoviska bez presunu paletky//
	IF Taktime_LeakageTestA_ST8A.CMD.START_Merania_2 THEN

		Milisekundy_2:= Milisekundy_2 + 4;//Pretože je v taskovej triede 4ms tak prirátaváme + 4//

		IF Milisekundy_2 >= 1000 THEN
			Sekundy_2:= Sekundy_2 + 1;
			Milisekundy_2:= 0;
		END_IF

		IF Sekundy_2 >= 60 THEN
			Minuty_2:= Minuty_2 + 1;
			Sekundy_2:= 0;
		END_IF

		IF Minuty_2 >= 60 THEN
			Hodiny_2:= Hodiny_2 + 1;
			Minuty_2:= 0;
		END_IF

	END_IF

	IF NOT Taktime_LeakageTestA_ST8A.CMD.START_Merania_2 THEN
		Milisekundy_2:= 0;
		Sekundy_2:= 0;
		Minuty_2:= 0;
		Hodiny_2:= 0;
	END_IF

	IF Taktime_LeakageTestA_ST8A.CMD.ZAPIS_Hodnot_2 THEN
		Taktime_LeakageTestA_ST8A.OUTPUTS.NameraneHodiny_2:= Hodiny_2;
		Taktime_LeakageTestA_ST8A.OUTPUTS.NameraneMinuty_2:= Minuty_2;
		Taktime_LeakageTestA_ST8A.OUTPUTS.NameraneSekundy_2:= Sekundy_2;
		Milisekundy_2:= 0;
		Sekundy_2:= 0;
		Minuty_2:= 0;
		Hodiny_2:= 0;
		Taktime_LeakageTestA_ST8A.CMD.ZAPIS_Hodnot_2:= FALSE;
	END_IF

	IF Taktime_LeakageTestA_ST8A.CMD.STOP_Merania_2 THEN
		Taktime_LeakageTestA_ST8A.OUTPUTS.NameraneHodiny_2:= Hodiny_2;
		Taktime_LeakageTestA_ST8A.OUTPUTS.NameraneMinuty_2:= Minuty_2;
		Taktime_LeakageTestA_ST8A.OUTPUTS.NameraneSekundy_2:= Sekundy_2;
		Taktime_LeakageTestA_ST8A.CMD.START_Merania_2:= FALSE;
		Taktime_LeakageTestA_ST8A.CMD.STOP_Merania_2:= FALSE;
	END_IF

END_PROGRAM

PROGRAM _EXIT
	(* Insert code here *)

END_PROGRAM
```

#### Variables.var - Local variables
```iecst
VAR
	Milisekundy_1 : UINT;
	Sekundy_1 : UINT;
	Minuty_1 : UINT;
	Hodiny_1 : UINT;
	Milisekundy_2 : UINT;
	Sekundy_2 : UINT;
	Minuty_2 : UINT;
	Hodiny_2 : UINT;
END_VAR
```

### Program Logical/MeranieTaktimePracovisk/Taktime_LeakageTestB_ST8B (IEC)

#### Main.st - Init, cyclic, exit code
```iecst
PROGRAM _INIT
	(* Insert code here *)

END_PROGRAM

PROGRAM _CYCLIC

        //Taktime pracoviska s presunom paletky//
	IF Taktime_LeakageTestB_ST8B.CMD.START_Merania_1 THEN

		Milisekundy_1:= Milisekundy_1 + 8;//Pretože je v taskovej triede 8ms tak prirátaváme + 8//

		IF Milisekundy_1 >= 1000 THEN
			Sekundy_1:= Sekundy_1 + 1;
			Milisekundy_1:= 0;
		END_IF

		IF Sekundy_1 >= 60 THEN
			Minuty_1:= Minuty_1 + 1;
			Sekundy_1:= 0;
		END_IF

		IF Minuty_1 >= 60 THEN
			Hodiny_1:= Hodiny_1 + 1;
			Minuty_1:= 0;
		END_IF

	END_IF

	IF NOT Taktime_LeakageTestB_ST8B.CMD.START_Merania_1 THEN
		Milisekundy_1:= 0;
		Sekundy_1:= 0;
		Minuty_1:= 0;
		Hodiny_1:= 0;
	END_IF

	IF Taktime_LeakageTestB_ST8B.CMD.ZAPIS_Hodnot_1 THEN
		Taktime_LeakageTestB_ST8B.OUTPUTS.NameraneHodiny_1:= Hodiny_1;
		Taktime_LeakageTestB_ST8B.OUTPUTS.NameraneMinuty_1:= Minuty_1;
		Taktime_LeakageTestB_ST8B.OUTPUTS.NameraneSekundy_1:= Sekundy_1;
		Milisekundy_1:= 0;
		Sekundy_1:= 0;
		Minuty_1:= 0;
		Hodiny_1:= 0;
		Taktime_LeakageTestB_ST8B.CMD.ZAPIS_Hodnot_1:= FALSE;
	END_IF

	IF Taktime_LeakageTestB_ST8B.CMD.STOP_Merania_1 THEN
		Taktime_LeakageTestB_ST8B.OUTPUTS.NameraneHodiny_1:= Hodiny_1;
		Taktime_LeakageTestB_ST8B.OUTPUTS.NameraneMinuty_1:= Minuty_1;
		Taktime_LeakageTestB_ST8B.OUTPUTS.NameraneSekundy_1:= Sekundy_1;
		Taktime_LeakageTestB_ST8B.CMD.START_Merania_1:= FALSE;
		Taktime_LeakageTestB_ST8B.CMD.STOP_Merania_1:= FALSE;
	END_IF

	//Taktime pracoviska bez presunu paletky//
	IF Taktime_LeakageTestB_ST8B.CMD.START_Merania_2 THEN

		Milisekundy_2:= Milisekundy_2 + 4;//Pretože je v taskovej triede 4ms tak prirátaváme + 4//

		IF Milisekundy_2 >= 1000 THEN
			Sekundy_2:= Sekundy_2 + 1;
			Milisekundy_2:= 0;
		END_IF

		IF Sekundy_2 >= 60 THEN
			Minuty_2:= Minuty_2 + 1;
			Sekundy_2:= 0;
		END_IF

		IF Minuty_2 >= 60 THEN
			Hodiny_2:= Hodiny_2 + 1;
			Minuty_2:= 0;
		END_IF

	END_IF

	IF NOT Taktime_LeakageTestB_ST8B.CMD.START_Merania_2 THEN
		Milisekundy_2:= 0;
		Sekundy_2:= 0;
		Minuty_2:= 0;
		Hodiny_2:= 0;
	END_IF

	IF Taktime_LeakageTestB_ST8B.CMD.ZAPIS_Hodnot_2 THEN
		Taktime_LeakageTestB_ST8B.OUTPUTS.NameraneHodiny_2:= Hodiny_2;
		Taktime_LeakageTestB_ST8B.OUTPUTS.NameraneMinuty_2:= Minuty_2;
		Taktime_LeakageTestB_ST8B.OUTPUTS.NameraneSekundy_2:= Sekundy_2;
		Milisekundy_2:= 0;
		Sekundy_2:= 0;
		Minuty_2:= 0;
		Hodiny_2:= 0;
		Taktime_LeakageTestB_ST8B.CMD.ZAPIS_Hodnot_2:= FALSE;
	END_IF

	IF Taktime_LeakageTestB_ST8B.CMD.STOP_Merania_2 THEN
		Taktime_LeakageTestB_ST8B.OUTPUTS.NameraneHodiny_2:= Hodiny_2;
		Taktime_LeakageTestB_ST8B.OUTPUTS.NameraneMinuty_2:= Minuty_2;
		Taktime_LeakageTestB_ST8B.OUTPUTS.NameraneSekundy_2:= Sekundy_2;
		Taktime_LeakageTestB_ST8B.CMD.START_Merania_2:= FALSE;
		Taktime_LeakageTestB_ST8B.CMD.STOP_Merania_2:= FALSE;
	END_IF

END_PROGRAM

PROGRAM _EXIT
	(* Insert code here *)

END_PROGRAM
```

#### Variables.var - Local variables
```iecst
VAR
	Milisekundy_1 : UINT;
	Sekundy_1 : UINT;
	Minuty_1 : UINT;
	Hodiny_1 : UINT;
	Milisekundy_2 : UINT;
	Sekundy_2 : UINT;
	Minuty_2 : UINT;
	Hodiny_2 : UINT;
END_VAR
```

### Program Logical/MeranieTaktimePracovisk/Taktime_FunkcnyTestA_ST9A (IEC)

#### Main.st - Init, cyclic, exit code
```iecst
PROGRAM _INIT
	(* Insert code here *)

END_PROGRAM

PROGRAM _CYCLIC

     //Taktime pracoviska s presunom paletky//
    IF Taktime_FunkcnyTestA.CMD.START_Merania_1 THEN

        Milisekundy_1:= Milisekundy_1 + 8;//Pretože je v taskovej triede 8ms tak prirátaváme + 8//

        IF Milisekundy_1 >= 1000 THEN
            Sekundy_1:= Sekundy_1 + 1;
            Milisekundy_1:= 0;
        END_IF

        IF Sekundy_1 >= 60 THEN
            Minuty_1:= Minuty_1 + 1;
            Sekundy_1:= 0;
        END_IF

        IF Minuty_1 >= 60 THEN
            Hodiny_1:= Hodiny_1 + 1;
            Minuty_1:= 0;
        END_IF

    END_IF

    IF NOT Taktime_FunkcnyTestA.CMD.START_Merania_1 THEN
        Milisekundy_1:= 0;
        Sekundy_1:= 0;
        Minuty_1:= 0;
        Hodiny_1:= 0;
    END_IF

    IF Taktime_FunkcnyTestA.CMD.ZAPIS_Hodnot_1 THEN
        Taktime_FunkcnyTestA.OUTPUTS.NameraneHodiny_1:= Hodiny_1;
        Taktime_FunkcnyTestA.OUTPUTS.NameraneMinuty_1:= Minuty_1;
        Taktime_FunkcnyTestA.OUTPUTS.NameraneSekundy_1:= Sekundy_1;
        Milisekundy_1:= 0;
        Sekundy_1:= 0;
        Minuty_1:= 0;
        Hodiny_1:= 0;
        Taktime_FunkcnyTestA.CMD.ZAPIS_Hodnot_1:= FALSE;
    END_IF

	IF Taktime_FunkcnyTestA.CMD.STOP_Merania_1 THEN
		Taktime_FunkcnyTestA.OUTPUTS.NameraneHodiny_1:= Hodiny_1;
		Taktime_FunkcnyTestA.OUTPUTS.NameraneMinuty_1:= Minuty_1;
		Taktime_FunkcnyTestA.OUTPUTS.NameraneSekundy_1:= Sekundy_1;
		Taktime_FunkcnyTestA.CMD.START_Merania_1:= FALSE;
		Taktime_FunkcnyTestA.CMD.STOP_Merania_1:= FALSE;
	END_IF

    //Taktime pracoviska bez presunu paletky//
    IF Taktime_FunkcnyTestA.CMD.START_Merania_2 THEN

        Milisekundy_2:= Milisekundy_2 + 4;//Pretože je v taskovej triede 4ms tak prirátaváme + 4//

        IF Milisekundy_2 >= 1000 THEN
            Sekundy_2:= Sekundy_2 + 1;
            Milisekundy_2:= 0;
        END_IF

        IF Sekundy_2 >= 60 THEN
            Minuty_2:= Minuty_2 + 1;
            Sekundy_2:= 0;
        END_IF

        IF Minuty_2 >= 60 THEN
            Hodiny_2:= Hodiny_2 + 1;
            Minuty_2:= 0;
        END_IF

    END_IF

    IF NOT Taktime_FunkcnyTestA.CMD.START_Merania_2 THEN
        Milisekundy_2:= 0;
        Sekundy_2:= 0;
        Minuty_2:= 0;
        Hodiny_2:= 0;
    END_IF

    IF Taktime_FunkcnyTestA.CMD.ZAPIS_Hodnot_2 THEN
        Taktime_FunkcnyTestA.OUTPUTS.NameraneHodiny_2:= Hodiny_2;
        Taktime_FunkcnyTestA.OUTPUTS.NameraneMinuty_2:= Minuty_2;
        Taktime_FunkcnyTestA.OUTPUTS.NameraneSekundy_2:= Sekundy_2;
        Milisekundy_2:= 0;
        Sekundy_2:= 0;
        Minuty_2:= 0;
        Hodiny_2:= 0;
        Taktime_FunkcnyTestA.CMD.ZAPIS_Hodnot_2:= FALSE;
    END_IF

	IF Taktime_FunkcnyTestA.CMD.STOP_Merania_2 THEN
		Taktime_FunkcnyTestA.OUTPUTS.NameraneHodiny_2:= Hodiny_2;
		Taktime_FunkcnyTestA.OUTPUTS.NameraneMinuty_2:= Minuty_2;
		Taktime_FunkcnyTestA.OUTPUTS.NameraneSekundy_2:= Sekundy_2;
		Taktime_FunkcnyTestA.CMD.START_Merania_2:= FALSE;
		Taktime_FunkcnyTestA.CMD.STOP_Merania_2:= FALSE;
	END_IF

END_PROGRAM

PROGRAM _EXIT
	(* Insert code here *)

END_PROGRAM
```

#### Variables.var - Local variables
```iecst
VAR
	Milisekundy_1 : UINT;
	Sekundy_1 : UINT;
	Minuty_1 : UINT;
	Hodiny_1 : UINT;
	Milisekundy_2 : UINT;
	Sekundy_2 : UINT;
	Minuty_2 : UINT;
	Hodiny_2 : UINT;
END_VAR
```

### Program Logical/MeranieTaktimePracovisk/Taktime_FunkcnyTestB_ST9B (IEC)

#### Main.st - Init, cyclic, exit code
```iecst
PROGRAM _INIT
	(* Insert code here *)

END_PROGRAM

PROGRAM _CYCLIC

    //Taktime pracoviska s presunom paletky//
    IF Taktime_FunkcnyTestB.CMD.START_Merania_1 THEN

        Milisekundy_1:= Milisekundy_1 + 8;//Pretože je v taskovej triede 8ms tak prirátaváme + 8//

        IF Milisekundy_1 >= 1000 THEN
            Sekundy_1:= Sekundy_1 + 1;
            Milisekundy_1:= 0;
        END_IF

        IF Sekundy_1 >= 60 THEN
            Minuty_1:= Minuty_1 + 1;
            Sekundy_1:= 0;
        END_IF

        IF Minuty_1 >= 60 THEN
            Hodiny_1:= Hodiny_1 + 1;
            Minuty_1:= 0;
        END_IF

    END_IF

    IF NOT Taktime_FunkcnyTestB.CMD.START_Merania_1 THEN
        Milisekundy_1:= 0;
        Sekundy_1:= 0;
        Minuty_1:= 0;
        Hodiny_1:= 0;
    END_IF

    IF Taktime_FunkcnyTestB.CMD.ZAPIS_Hodnot_1 THEN
        Taktime_FunkcnyTestB.OUTPUTS.NameraneHodiny_1:= Hodiny_1;
        Taktime_FunkcnyTestB.OUTPUTS.NameraneMinuty_1:= Minuty_1;
        Taktime_FunkcnyTestB.OUTPUTS.NameraneSekundy_1:= Sekundy_1;
        Milisekundy_1:= 0;
        Sekundy_1:= 0;
        Minuty_1:= 0;
        Hodiny_1:= 0;
        Taktime_FunkcnyTestB.CMD.ZAPIS_Hodnot_1:= FALSE;
    END_IF

	IF Taktime_FunkcnyTestB.CMD.STOP_Merania_1 THEN
		Taktime_FunkcnyTestB.OUTPUTS.NameraneHodiny_1:= Hodiny_1;
		Taktime_FunkcnyTestB.OUTPUTS.NameraneMinuty_1:= Minuty_1;
		Taktime_FunkcnyTestB.OUTPUTS.NameraneSekundy_1:= Sekundy_1;
		Taktime_FunkcnyTestB.CMD.START_Merania_1:= FALSE;
		Taktime_FunkcnyTestB.CMD.STOP_Merania_1:= FALSE;
	END_IF

    //Taktime pracoviska bez presunu paletky//
    IF Taktime_FunkcnyTestB.CMD.START_Merania_2 THEN

        Milisekundy_2:= Milisekundy_2 + 4;//Pretože je v taskovej triede 4ms tak prirátaváme + 4//

        IF Milisekundy_2 >= 1000 THEN
            Sekundy_2:= Sekundy_2 + 1;
            Milisekundy_2:= 0;
        END_IF

        IF Sekundy_2 >= 60 THEN
            Minuty_2:= Minuty_2 + 1;
            Sekundy_2:= 0;
        END_IF

        IF Minuty_2 >= 60 THEN
            Hodiny_2:= Hodiny_2 + 1;
            Minuty_2:= 0;
        END_IF

    END_IF

    IF NOT Taktime_FunkcnyTestB.CMD.START_Merania_2 THEN
        Milisekundy_2:= 0;
        Sekundy_2:= 0;
        Minuty_2:= 0;
        Hodiny_2:= 0;
    END_IF

    IF Taktime_FunkcnyTestB.CMD.ZAPIS_Hodnot_2 THEN
        Taktime_FunkcnyTestB.OUTPUTS.NameraneHodiny_2:= Hodiny_2;
        Taktime_FunkcnyTestB.OUTPUTS.NameraneMinuty_2:= Minuty_2;
        Taktime_FunkcnyTestB.OUTPUTS.NameraneSekundy_2:= Sekundy_2;
        Milisekundy_2:= 0;
        Sekundy_2:= 0;
        Minuty_2:= 0;
        Hodiny_2:= 0;
        Taktime_FunkcnyTestB.CMD.ZAPIS_Hodnot_2:= FALSE;
    END_IF

	IF Taktime_FunkcnyTestB.CMD.STOP_Merania_2 THEN
		Taktime_FunkcnyTestB.OUTPUTS.NameraneHodiny_2:= Hodiny_2;
		Taktime_FunkcnyTestB.OUTPUTS.NameraneMinuty_2:= Minuty_2;
		Taktime_FunkcnyTestB.OUTPUTS.NameraneSekundy_2:= Sekundy_2;
		Taktime_FunkcnyTestB.CMD.START_Merania_2:= FALSE;
		Taktime_FunkcnyTestB.CMD.STOP_Merania_2:= FALSE;
	END_IF

END_PROGRAM

PROGRAM _EXIT
	(* Insert code here *)

END_PROGRAM
```

#### Variables.var - Local variables
```iecst
VAR
	Milisekundy_1 : UINT;
	Sekundy_1 : UINT;
	Minuty_1 : UINT;
	Hodiny_1 : UINT;
	Milisekundy_2 : UINT;
	Sekundy_2 : UINT;
	Minuty_2 : UINT;
	Hodiny_2 : UINT;
END_VAR
```

### Program Logical/MeranieTaktimePracovisk/Taktime_Etiketovacka_ST9 (IEC)

#### Main.st - Init, cyclic, exit code
```iecst
PROGRAM _INIT
	(* Insert code here *)

END_PROGRAM

PROGRAM _CYCLIC

     //Taktime pracoviska s presunom paletky//
    IF Taktime_Etiketovacka_ST9.CMD.START_Merania_1 THEN

        Milisekundy_1:= Milisekundy_1 + 8;//Pretože je v taskovej triede 8ms tak prirátaváme + 8//

        IF Milisekundy_1 >= 1000 THEN
            Sekundy_1:= Sekundy_1 + 1;
            Milisekundy_1:= 0;
        END_IF

        IF Sekundy_1 >= 60 THEN
            Minuty_1:= Minuty_1 + 1;
            Sekundy_1:= 0;
        END_IF

        IF Minuty_1 >= 60 THEN
            Hodiny_1:= Hodiny_1 + 1;
            Minuty_1:= 0;
        END_IF

    END_IF

    IF NOT Taktime_Etiketovacka_ST9.CMD.START_Merania_1 THEN
        Milisekundy_1:= 0;
        Sekundy_1:= 0;
        Minuty_1:= 0;
        Hodiny_1:= 0;
    END_IF

    IF Taktime_Etiketovacka_ST9.CMD.ZAPIS_Hodnot_1 THEN
        Taktime_Etiketovacka_ST9.OUTPUTS.NameraneHodiny_1:= Hodiny_1;
        Taktime_Etiketovacka_ST9.OUTPUTS.NameraneMinuty_1:= Minuty_1;
        Taktime_Etiketovacka_ST9.OUTPUTS.NameraneSekundy_1:= Sekundy_1;
        Milisekundy_1:= 0;
        Sekundy_1:= 0;
        Minuty_1:= 0;
        Hodiny_1:= 0;
        Taktime_Etiketovacka_ST9.CMD.ZAPIS_Hodnot_1:= FALSE;
    END_IF

	IF Taktime_Etiketovacka_ST9.CMD.STOP_Merania_1 THEN
		Taktime_Etiketovacka_ST9.OUTPUTS.NameraneHodiny_1:= Hodiny_1;
		Taktime_Etiketovacka_ST9.OUTPUTS.NameraneMinuty_1:= Minuty_1;
		Taktime_Etiketovacka_ST9.OUTPUTS.NameraneSekundy_1:= Sekundy_1;
		Taktime_Etiketovacka_ST9.CMD.START_Merania_1:= FALSE;
		Taktime_Etiketovacka_ST9.CMD.STOP_Merania_1:= FALSE;
	END_IF

    //Taktime pracoviska bez presunu paletky//
    IF Taktime_Etiketovacka_ST9.CMD.START_Merania_2 THEN

        Milisekundy_2:= Milisekundy_2 + 4;//Pretože je v taskovej triede 4ms tak prirátaváme + 4//

        IF Milisekundy_2 >= 1000 THEN
            Sekundy_2:= Sekundy_2 + 1;
            Milisekundy_2:= 0;
        END_IF

        IF Sekundy_2 >= 60 THEN
            Minuty_2:= Minuty_2 + 1;
            Sekundy_2:= 0;
        END_IF

        IF Minuty_2 >= 60 THEN
            Hodiny_2:= Hodiny_2 + 1;
            Minuty_2:= 0;
        END_IF

    END_IF

    IF NOT Taktime_Etiketovacka_ST9.CMD.START_Merania_2 THEN
        Milisekundy_2:= 0;
        Sekundy_2:= 0;
        Minuty_2:= 0;
        Hodiny_2:= 0;
    END_IF

    IF Taktime_Etiketovacka_ST9.CMD.ZAPIS_Hodnot_2 THEN
        Taktime_Etiketovacka_ST9.OUTPUTS.NameraneHodiny_2:= Hodiny_2;
        Taktime_Etiketovacka_ST9.OUTPUTS.NameraneMinuty_2:= Minuty_2;
        Taktime_Etiketovacka_ST9.OUTPUTS.NameraneSekundy_2:= Sekundy_2;
        Milisekundy_2:= 0;
        Sekundy_2:= 0;
        Minuty_2:= 0;
        Hodiny_2:= 0;
        Taktime_Etiketovacka_ST9.CMD.ZAPIS_Hodnot_2:= FALSE;
    END_IF

	IF Taktime_Etiketovacka_ST9.CMD.STOP_Merania_2 THEN
		Taktime_Etiketovacka_ST9.OUTPUTS.NameraneHodiny_2:= Hodiny_2;
		Taktime_Etiketovacka_ST9.OUTPUTS.NameraneMinuty_2:= Minuty_2;
		Taktime_Etiketovacka_ST9.OUTPUTS.NameraneSekundy_2:= Sekundy_2;
		Taktime_Etiketovacka_ST9.CMD.START_Merania_2:= FALSE;
		Taktime_Etiketovacka_ST9.CMD.STOP_Merania_2:= FALSE;
	END_IF

END_PROGRAM

PROGRAM _EXIT
	(* Insert code here *)

END_PROGRAM
```

#### Variables.var - Local variables
```iecst
VAR
	Milisekundy_1 : UINT;
	Sekundy_1 : UINT;
	Minuty_1 : UINT;
	Hodiny_1 : UINT;
	Milisekundy_2 : UINT;
	Sekundy_2 : UINT;
	Minuty_2 : UINT;
	Hodiny_2 : UINT;
END_VAR
```

### Program Logical/MeranieTaktimePracovisk/Taktime_Vytah_ST10 (IEC)

#### Main.st - Init, cyclic, exit code
```iecst
PROGRAM _INIT
	(* Insert code here *)

END_PROGRAM

PROGRAM _CYCLIC
	 //Taktime pracoviska s presunom paletky//
    IF Taktime_Vytah_ST10.CMD.START_Merania_1 THEN

        Milisekundy_1:= Milisekundy_1 + 8;//Pretože je v taskovej triede 8ms tak prirátaváme + 8//

        IF Milisekundy_1 >= 1000 THEN
            Sekundy_1:= Sekundy_1 + 1;
            Milisekundy_1:= 0;
        END_IF

        IF Sekundy_1 >= 60 THEN
            Minuty_1:= Minuty_1 + 1;
            Sekundy_1:= 0;
        END_IF

        IF Minuty_1 >= 60 THEN
            Hodiny_1:= Hodiny_1 + 1;
            Minuty_1:= 0;
        END_IF

    END_IF

    IF NOT Taktime_Vytah_ST10.CMD.START_Merania_1 THEN
        Milisekundy_1:= 0;
        Sekundy_1:= 0;
        Minuty_1:= 0;
        Hodiny_1:= 0;
    END_IF

    IF Taktime_Vytah_ST10.CMD.ZAPIS_Hodnot_1 THEN
        Taktime_Vytah_ST10.OUTPUTS.NameraneHodiny_1:= Hodiny_1;
        Taktime_Vytah_ST10.OUTPUTS.NameraneMinuty_1:= Minuty_1;
        Taktime_Vytah_ST10.OUTPUTS.NameraneSekundy_1:= Sekundy_1;
        Milisekundy_1:= 0;
        Sekundy_1:= 0;
        Minuty_1:= 0;
        Hodiny_1:= 0;
        Taktime_Vytah_ST10.CMD.ZAPIS_Hodnot_1:= FALSE;
    END_IF

	IF Taktime_Vytah_ST10.CMD.STOP_Merania_1 THEN
		Taktime_Vytah_ST10.OUTPUTS.NameraneHodiny_1:= Hodiny_1;
		Taktime_Vytah_ST10.OUTPUTS.NameraneMinuty_1:= Minuty_1;
		Taktime_Vytah_ST10.OUTPUTS.NameraneSekundy_1:= Sekundy_1;
		Taktime_Vytah_ST10.CMD.START_Merania_1:= FALSE;
		Taktime_Vytah_ST10.CMD.STOP_Merania_1:= FALSE;
	END_IF

    //Taktime pracoviska bez presunu paletky//
    IF Taktime_Vytah_ST10.CMD.START_Merania_2 THEN

        Milisekundy_2:= Milisekundy_2 + 4;//Pretože je v taskovej triede 4ms tak prirátaváme + 4//

        IF Milisekundy_2 >= 1000 THEN
            Sekundy_2:= Sekundy_2 + 1;
            Milisekundy_2:= 0;
        END_IF

        IF Sekundy_2 >= 60 THEN
            Minuty_2:= Minuty_2 + 1;
            Sekundy_2:= 0;
        END_IF

        IF Minuty_2 >= 60 THEN
            Hodiny_2:= Hodiny_2 + 1;
            Minuty_2:= 0;
        END_IF

    END_IF

    IF NOT Taktime_Vytah_ST10.CMD.START_Merania_2 THEN
        Milisekundy_2:= 0;
        Sekundy_2:= 0;
        Minuty_2:= 0;
        Hodiny_2:= 0;
    END_IF

    IF Taktime_Vytah_ST10.CMD.ZAPIS_Hodnot_2 THEN
        Taktime_Vytah_ST10.OUTPUTS.NameraneHodiny_2:= Hodiny_2;
        Taktime_Vytah_ST10.OUTPUTS.NameraneMinuty_2:= Minuty_2;
        Taktime_Vytah_ST10.OUTPUTS.NameraneSekundy_2:= Sekundy_2;
        Milisekundy_2:= 0;
        Sekundy_2:= 0;
        Minuty_2:= 0;
        Hodiny_2:= 0;
        Taktime_Vytah_ST10.CMD.ZAPIS_Hodnot_2:= FALSE;
    END_IF

	IF Taktime_Vytah_ST10.CMD.STOP_Merania_2 THEN
		Taktime_Vytah_ST10.OUTPUTS.NameraneHodiny_2:= Hodiny_2;
		Taktime_Vytah_ST10.OUTPUTS.NameraneMinuty_2:= Minuty_2;
		Taktime_Vytah_ST10.OUTPUTS.NameraneSekundy_2:= Sekundy_2;
		Taktime_Vytah_ST10.CMD.START_Merania_2:= FALSE;
		Taktime_Vytah_ST10.CMD.STOP_Merania_2:= FALSE;
	END_IF

END_PROGRAM

PROGRAM _EXIT
	(* Insert code here *)

END_PROGRAM
```

#### Variables.var - Local variables
```iecst
VAR
	Milisekundy_1 : UINT;
	Sekundy_1 : UINT;
	Minuty_1 : UINT;
	Hodiny_1 : UINT;
	Milisekundy_2 : UINT;
	Sekundy_2 : UINT;
	Minuty_2 : UINT;
	Hodiny_2 : UINT;
END_VAR
```

### RecipeGlobal.typ - Global data types
```iecst
(************************************************************************Receptury****************************************************)

TYPE
	recSTATE :
		( (*Recipe managment state machine*)
		REC_WAIT,
		REC_REG_NAME,
		REC_REG_VAR,
		REC_CREATE_DIR,
		REC_READ_DIR,
		REC_READ_DIR_1,
		REC_READ_DIR_2,
		REC_READ_DIR_3,
		REC_GEN_FILE_NAME,
		REC_LOAD_SAVE,
		REC_DELETE,
		REC_RENAME,
		REC_ERROR
		);
	recTYPE :
		( (*Typ súboru do ktorého sa budú receptury ukladať*)
		typeCSV,
		typeXML
		);
	recERR : 	STRUCT  (*Recipe managment error structure*)
		Text : WSTRING[200]; (* Error text *)
		No : DINT; (* Error number *)
		State : recSTATE; (* Error step *)
	END_STRUCT;
	recCMD : 	STRUCT  (*Recipe managment command structure*)
		Init : BOOL := TRUE;
		New : BOOL;
		Load : BOOL;
		Save : BOOL;
		Rename : BOOL;
		Delete : BOOL; (* Delete selected file *)
		ErrorReset : BOOL;
	END_STRUCT;
	recPAR : 	STRUCT  (*Recipe managment parameter structure*)
		RecipeVariable : STRING[200]; (*Name of the variable where the data is stored*)
		RecipeName : WSTRING[REC_NAME_LENGTH]; (*Recipe name*)
		RecipeNameNew : WSTRING[REC_NAME_LENGTH]; (*Recipe name*)
		RecipeID : STRING[REC_NAME_LENGTH]; (*Recipe name*)
		RecipeDirectory : STRING[200]; (*Recipe directory*)
		DeviceName : STRING[100]; (*Device name where the recipes are stored*)
		MpLink : MpComIdentType; (*MpLink from mappRecipe*)
		Initialized : BOOL; (*Indicates that recipe managment was initialized*)
		VisuSlotID : USINT; (*ID for connected web connection*)
		VisuEnableCommand : BOOL;
	END_STRUCT;
	recDAT : 	STRUCT  (*Recipe managment data structure*)
		RecipeNames : ARRAY[0..REC_MAX_NUM]OF WSTRING[REC_NAME_LENGTH]; (*Recipe unicode name*)
		RecipeIDs : ARRAY[0..REC_MAX_NUM]OF STRING[REC_NAME_LENGTH]; (*Recipe unicode name*)
		RecipeNum : UINT; (*Number of recipes*)
		Status : WSTRING[100]; (*Shows the result of the last command*)
	END_STRUCT;
	recVIS : 	STRUCT  (*Recipe managment visualization structure*)
		RecipeNames : ARRAY[0..REC_MAX_NUM]OF WSTRING[REC_VIS_LENGTH]; (*Recipe file size*)
		RecipeNum : UINT; (*Number of recipes*)
		RecipeFilter : WSTRING[REC_NAME_LENGTH]; (*Filter for recipe name	*)
		RecipeSelect : WSTRING[REC_NAME_LENGTH]; (*Select new or renamed recipe in list box*)
		ShowMessageBoxError : BOOL; (*Show message box on error*)
	END_STRUCT;
	recMAIN : 	STRUCT  (*Recipe managment main structure*)
		CMD : recCMD; (* Command structure *)
		PAR : recPAR; (* Parameter structure *)
		DAT : recDAT; (*Data structure*)
		VIS : ARRAY[0..REC_MAX_CLIENTS_ID]OF recVIS; (*Visualization structure*)
		ERR : recERR; (* Error structure *)
	END_STRUCT;
	recVariable : 	STRUCT  (*Premenné receptur*)
		Temperature1 : INT := 11;
		Temperature2 : INT := 22;
		MotorSpeed : DINT := 33;
		Position : REAL := 44.55;
	END_STRUCT;
END_TYPE
```

### RecipeGlobal.var - Global variables
```iecst
VAR CONSTANT
	REC_USE_UNICODE : BOOL := TRUE; (*Use standard strings for recipe name when false, use unicode strings for recipe name when true*)
END_VAR
VAR
	REC_RECIPE_TYPE : recTYPE := typeCSV; (*Type of recipe (CSV / XML), ak necháme volbu typeCSV bude zapisovať do súboru CSV ak nedáme volbu typeCSV bude zapisovať do súboru XML*)
END_VAR
VAR CONSTANT
	REC_MAX_NUM : USINT := 100; (*Maximálny počet receptur*)
	REC_NAME_LENGTH : USINT := 40; (*Maximálna dĺžka jména receptury*)
	REC_VIS_LENGTH : USINT := 120; (*Make this REC_NAME_LENGTH  x3*)
	REC_MAX_CLIENTS_ID : USINT := 2; (*Highest client ID for concurrent web client connections. Do not change this number.*)
END_VAR
VAR
	Recipe_01 : recMAIN; (*Global recipe structure. The name must match the task name of the recipe managment.*)
	RecipeData : recVariable; (*Data uložené v recepture*)
	EditaciaReceptur_ENABLE : BOOL;
END_VAR
```

### Program Logical/Receptury/Recipe_01 (IEC)
